FUNCTION_BLOCK NeredaCAeration (* Composite Function Block Type *)
  (* Standard: 61499-2 *)
  (* Version 0.0, 4/25/2024, SESA713705, Schneider Electric, template *)
  PACKAGE SE.Nereda;
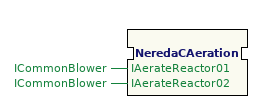
  SOCKETS
    IAerateReactor01 : ICommonBlower;
    IAerateReactor02 : ICommonBlower;
  END_SOCKETS
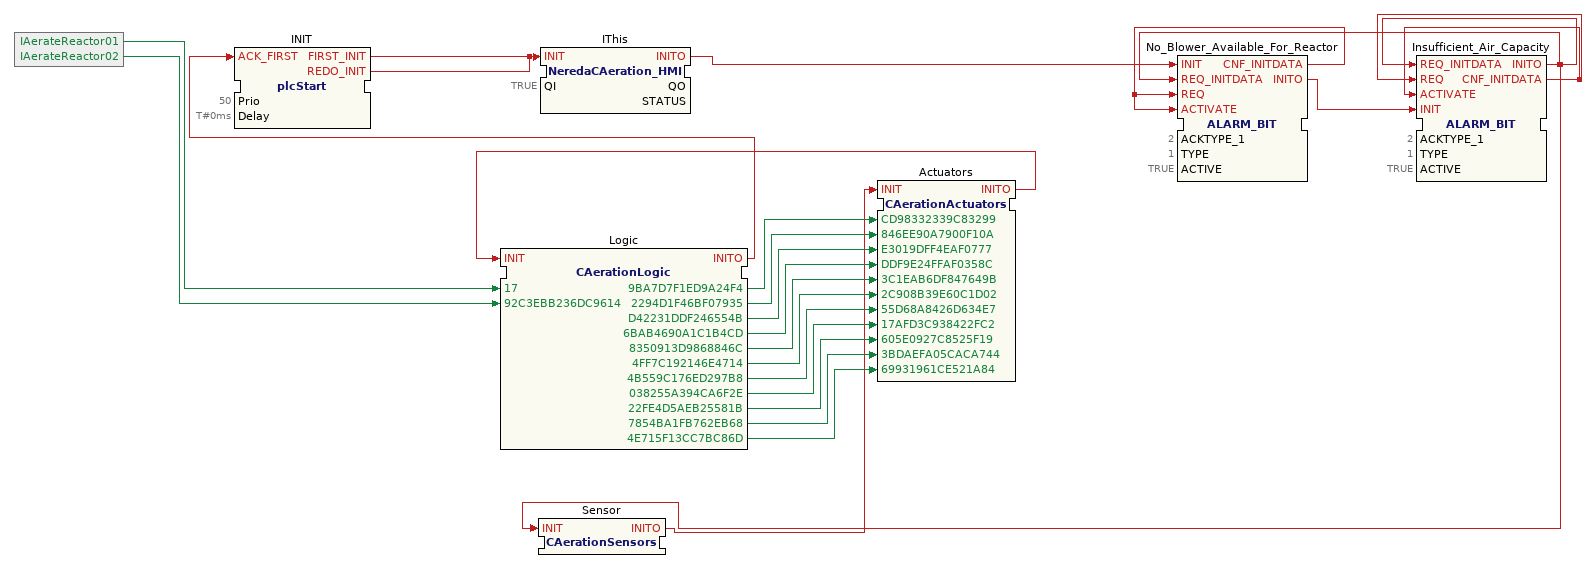
  (* 01 - FUNCTIONNAL INPUT INTERFACE *)
  (* 00 - INITIALIZATION *)
  (* 05 - LOGIC *)
  (* 06 - HMI INTERFACE *)
  (* 03 - FIELD INTERFACE *)
  (* 02 - FUNCTIONNAL OUTPUT INTERFACE *)
  (* Aeartion Logic *)
  (* 04 - CHILDREN *)
  (* 4A - TYPICALS *)
  (* 07- REACTOR ALARM *)
  FBS
    Logic : CAerationLogic;
    IThis : NeredaCAeration_HMI(QI := TRUE);
    INIT : plcStart(Prio := 50, Delay := T#0ms);
    Sensor : CAerationSensors;
    No_Blower_Available_For_Reactor : ALARM_BIT(ACKTYPE_1 := 2, TYPE := 1, ACTIVE := TRUE);
    Insufficient_Air_Capacity : ALARM_BIT(ACKTYPE_1 := 2, TYPE := 1, ACTIVE := TRUE);
    Actuators : CAerationActuators; {SET_ATTRIBUTE(Configuration.Component.HideUnusedPorts, )}
  END_FBS
  EVENT_CONNECTIONS
    INIT.FIRST_INIT TO IThis.INIT;
    IThis.INITO TO No_Blower_Available_For_Reactor.INIT;
    Insufficient_Air_Capacity.INITO TO No_Blower_Available_For_Reactor.REQ_INITDATA;
    No_Blower_Available_For_Reactor.CNF_INITDATA TO No_Blower_Available_For_Reactor.REQ;
    INIT.REDO_INIT TO IThis.INIT;
    No_Blower_Available_For_Reactor.CNF_INITDATA TO No_Blower_Available_For_Reactor.ACTIVATE;
    Insufficient_Air_Capacity.INITO TO Sensor.INIT;
    Sensor.INITO TO Actuators.INIT;
    Logic.INITO TO INIT.ACK_FIRST;
    Insufficient_Air_Capacity.INITO TO Insufficient_Air_Capacity.REQ_INITDATA;
    Insufficient_Air_Capacity.CNF_INITDATA TO Insufficient_Air_Capacity.REQ;
    Insufficient_Air_Capacity.CNF_INITDATA TO Insufficient_Air_Capacity.ACTIVATE;
    No_Blower_Available_For_Reactor.INITO TO Insufficient_Air_Capacity.INIT;
    Actuators.INITO TO Logic.INIT;
  END_CONNECTIONS
  ADAPTER_CONNECTIONS
    IAerateReactor01 TO Logic.17;
    IAerateReactor02 TO Logic.92C3EBB236DC9614;
    Logic.9BA7D7F1ED9A24F4 TO Actuators.CD98332339C83299;
    Logic.2294D1F46BF07935 TO Actuators.846EE90A7900F10A;
    Logic.D42231DDF246554B TO Actuators.E3019DFF4EAF0777;
    Logic.6BAB4690A1C1B4CD TO Actuators.DDF9E24FFAF0358C;
    Logic.8350913D9868846C TO Actuators.3C1EAB6DF847649B;
    Logic.4FF7C192146E4714 TO Actuators.2C908B39E60C1D02;
    Logic.4B559C176ED297B8 TO Actuators.55D68A8426D634E7;
    Logic.038255A394CA6F2E TO Actuators.17AFD3C938422FC2;
    Logic.22FE4D5AEB25581B TO Actuators.605E0927C8525F19;
    Logic.7854BA1FB762EB68 TO Actuators.3BDAEFA05CACA744;
    Logic.4E715F13CC7BC86D TO Actuators.69931961CE521A84;
  END_CONNECTIONS
END_FUNCTION_BLOCK
